(* Logix 5000 project; controller cal1615 1756-L62 rev 20.19; software revision 20.05; part 61 of 82 *)
(* tags used below, declared in another part *)
   aaa_eb_temp2 : BOOL;
   FAULT : BOOL;   // Fault AFI
   p01_recipe_active : recipe;   // Active Recipe
   p01r02_plc_scan_time_in_sec : REAL;   // System PLC Scan Time in Seconds
   p01r09_pb_global_reset : BOOL;   // System Modes PB: Global Fault Reset
   p01r09_request_line_jog : BOOL;   // System Modes Request Line Jog Forward
   p01r09_stretch_mode : BOOL;
   p01r12_master_ramped_speed : REAL;   // System Line Accel Decel Control Master Ramped Speed
   p01r13_line_running : BOOL;   // System Line Start Sequence Line Running
   p01r13_line_slow_ramp : BOOL;   // System Line Start Sequence Start Line to Slow Speed
   p01r13_permissive_drives : BOOL;   // System Line Start Sequence Permissive Drives
   p01r13_state : DINT;   // System Line Start Sequence Sequencer Step
   p02_real_from_hmi : hmi_real;   // MOP HMI Iface Real from HMI
   p20r15_loa_on : BOOL;   // Letoff Letoff A VFD On
   p20r16_lob_on : BOOL;   // Letoff Letoff B On
   p22r09_mode_thread : BOOL;   // Tension Stand 1 Modes Thread Mode
   p22r10_pid_psn : PID;   // Tension Stand 1 Speed Tension PID Dancer Position
   p25_ai_speed : REAL;   // Tension Stand 2 Inputs Sufrace Speed [fpm]
   p25_ai_torque : REAL;
   p25_ai_ts2_lc : REAL;   // System Metering Roll VFD Minimum Start Tension
   p25_ao_selected_speed : REAL;   // Tension Stand 2 VFD Selected Speed
   p25_ao_torque : REAL;
   p25_control_word : INT;
   p25_di_brake : BOOL;   // Tension Stand 2 Digital Input TS2 & Slitter Brake Temperature OK
   p25_di_therm : BOOL;   // Tension Stand 2 Digital Input Motor Temperature OK
   p25_param_ts2_jog_speed : REAL;   // System Parameter Tension Stand 2 Jog Speed
   p25_status_word : INT;
   p25_ts2_acc_rate : REAL;
   p25_ts2_decel_rate : REAL;
   p25_ts2_vfd : ABB_PROTOCOL_VFD;
   p25r01 : routine;
   p25r02_tension_dev_max : REAL;
   p25r02_tension_dev_min : REAL;
   p25r09_mode_jog : BOOL;   // Tension Stand 2 Modes Jog Mode
   p25r09_mode_thread : BOOL;   // Tension Stand 2 Modes Thread Mode
   p25r09_pb_jog_fwd : BOOL;   // Tension Stand 2 Modes PB: Jog Forward
   p25r09_pb_jog_rev : BOOL;   // Tension Stand 2 Modes PB: Jog Reverse
   p25r10 : routine;
   p25r10_calc_speed_offset : REAL;
   p25r10_param_psn_gain : REAL;   // Tension Stand 2 Parameter Position Gain
   p25r10_pid_manual_request : BOOL;
   p25r10_pid_out : REAL;
   p25r10_pid_psn : PID;   // Tension Stand 2 Speed Tension PID Dancer Position Process Variable
   p25r10_pid_psn_cv : REAL;
   p25r10_pid_psn_pv : REAL;   // Tension Stand 2 Speed Tension PID Dancer Position Process Variable
   p25r10_speed_offset : REAL;   // Tension Stand 2 Speed tension Speed Offset from Base
   p25r10_tension_request : BOOL;
   p25r10_timer_fault : TIMER[4];   // Tension Stand 2 Speed Tension Fault Dwell Timer
   p25r10_timer_warning : TIMER[4];   // Tension Stand 2 Speed Tension Warning Dwell Timer
   p25r11 : routine;   // Tension Stand 2 VFD
   p25r11_acc_decel_ramp : SYS_ACC_DEC_RAMP;   // Tension Stand 2 VFD Accel /Decel Ramp
   p25r11_at_zero : BOOL;   // Tension Stand 2 VFD At Zero Speed
   p25r11_permissive_jog_thread : BOOL;   // Tension Stand 2 VFD Permissive Jog/Thread
   p25r11_request_jog_fwd : BOOL;   // Tension Stand 2 VFD Request Jog FWD
   p25r11_request_jog_rev : BOOL;   // Tension Stand 2 VFD Request Jog REV
   p25r11_request_line_jog : BOOL;   // Tension Stand 2 VFD Request Line Jog
   p25r11_request_line_run : BOOL;   // Tension Stant 2 VFD Request Line Run
   p25r11_request_thread_fwd : BOOL;   // Tension Stand 2 VFD Request Thread FWD
   p25r11_request_thread_rev : BOOL;   // Tension Stand 2 VFD Request Thread REV
   p25r11_selected_speed : REAL;   // Tension Stand 2 VFD Selected Speed
   p25r11_timer_fault : TIMER[10];   // Tension Stand 2 VFD Fault Dwell Timer
   p25r11_timer_warning : TIMER[4];   // Tension Stand VFD Warning Dwell Timer
   p25r11_vfd_start_request : BOOL;
   p29r15 : routine;   // Winder Winder A VFD
(* P25_Tension_Stand_2, continued *)

ROUTINE R10_Speed_Control   (* ladder *)
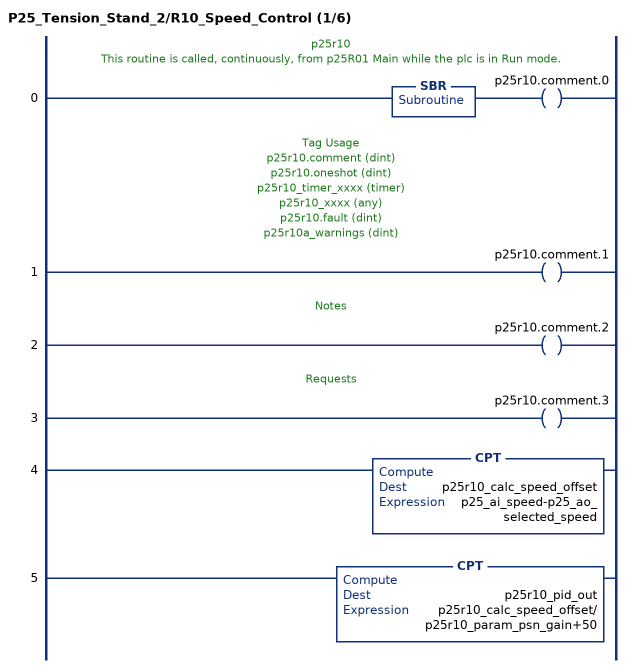
   // p25r10
   // This routine is called, continuously, from p25R01 Main while the plc is in Run mode.
   0: SBR()OTE(p25r10.comment.0);
   // Tag Usage
   // p25r10.comment (dint)
   // p25r10.oneshot (dint)
   // p25r10_timer_xxxx (timer)
   // p25r10_xxxx (any)
   // p25r10.fault (dint)
   // p25r10a_warnings (dint)
   1: OTE(p25r10.comment.1);
   // Notes
   2: OTE(p25r10.comment.2);
   // Requests
   3: OTE(p25r10.comment.3);
   4: CPT(p25r10_calc_speed_offset,p25_ai_speed-p25_ao_selected_speed);
   5: CPT(p25r10_pid_out,p25r10_calc_speed_offset/p25r10_param_psn_gain+50);
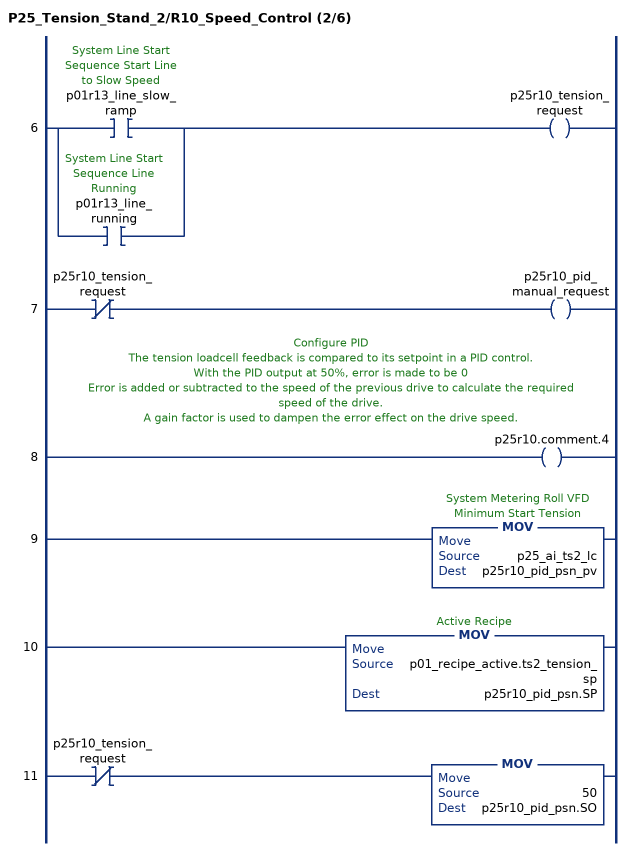
   6: [XIC(p01r13_line_slow_ramp) ,XIC(p01r13_line_running) ]OTE(p25r10_tension_request);
   7: XIO(p25r10_tension_request)OTE(p25r10_pid_manual_request);
   // Configure PID
   // The tension loadcell feedback is compared to its setpoint in a PID control.
   // With the PID output at 50%, error is made to be 0
   // Error is added or subtracted to the speed of the previous drive to calculate the required speed of the drive.
   // A gain factor is used to dampen the error effect on the drive speed.
   8: OTE(p25r10.comment.4);
   9: MOV(p25_ai_ts2_lc,p25r10_pid_psn_pv);
   10: MOV(p01_recipe_active.ts2_tension_sp,p25r10_pid_psn.SP);
   11: XIO(p25r10_tension_request)MOV(50,p25r10_pid_psn.SO);
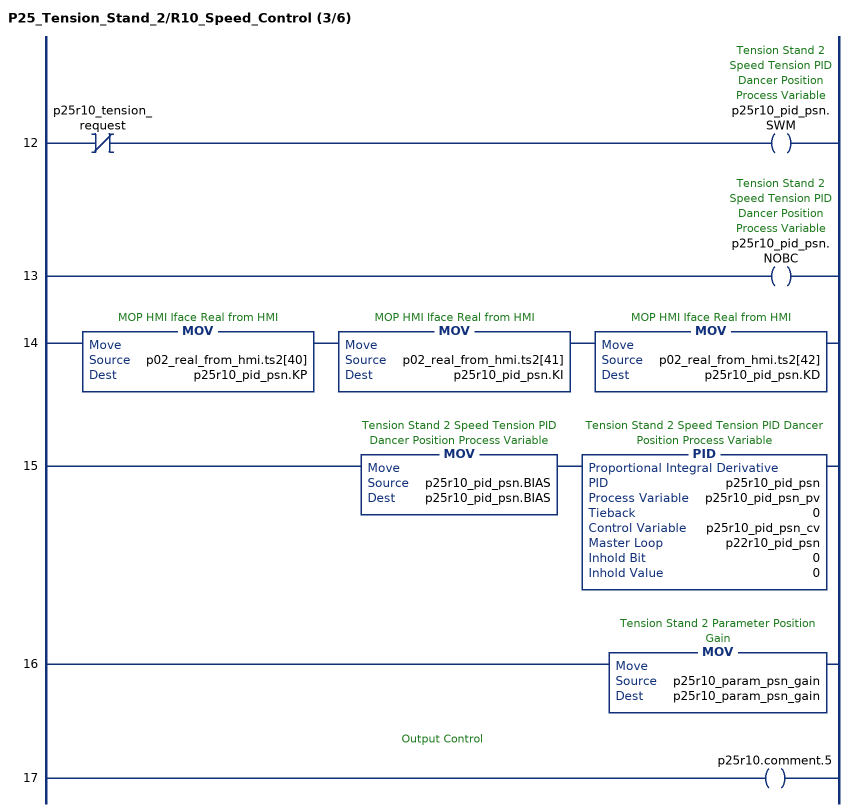
   12: XIO(p25r10_tension_request)OTE(p25r10_pid_psn.SWM);
   13: OTE(p25r10_pid_psn.NOBC);
   14: MOV(p02_real_from_hmi.ts2[40],p25r10_pid_psn.KP)MOV(p02_real_from_hmi.ts2[41],p25r10_pid_psn.KI)MOV(p02_real_from_hmi.ts2[42],p25r10_pid_psn.KD);
   15: MOV(p25r10_pid_psn.BIAS,p25r10_pid_psn.BIAS)PID(p25r10_pid_psn,p25r10_pid_psn_pv,0,p25r10_pid_psn_cv,p22r10_pid_psn,0,0);
   16: MOV(p25r10_param_psn_gain,p25r10_param_psn_gain);
   // Output Control
   17: OTE(p25r10.comment.5);
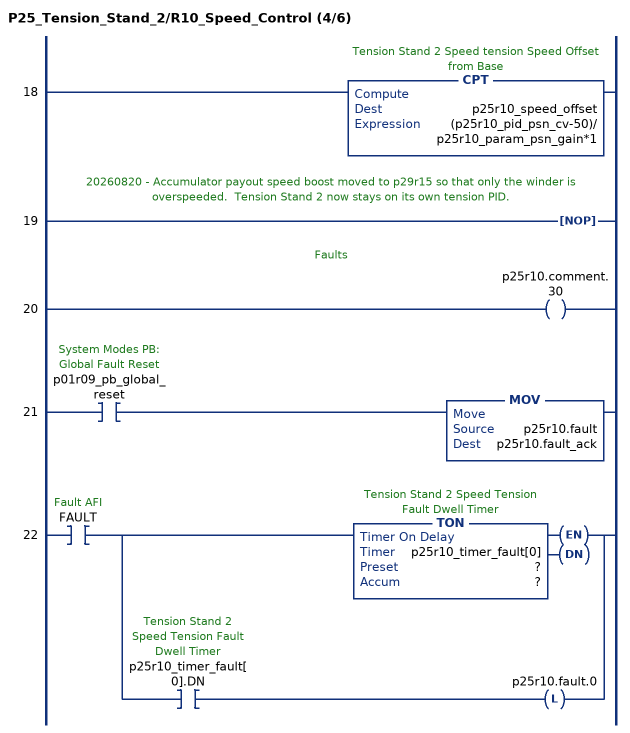
   18: CPT(p25r10_speed_offset,(p25r10_pid_psn_cv-50)/p25r10_param_psn_gain*1);
   // 20260820 - Accumulator payout speed boost moved to p29r15 so that only the winder is overspeeded.  Tension Stand 2 now stays on its own tension PID.
   19: NOP();
   // Faults
   20: OTE(p25r10.comment.30);
   21: XIC(p01r09_pb_global_reset)MOV(p25r10.fault,p25r10.fault_ack);
   22: XIC(FAULT)[TON(p25r10_timer_fault[0],?,?) ,XIC(p25r10_timer_fault[0].DN) OTL(p25r10.fault.0) ];
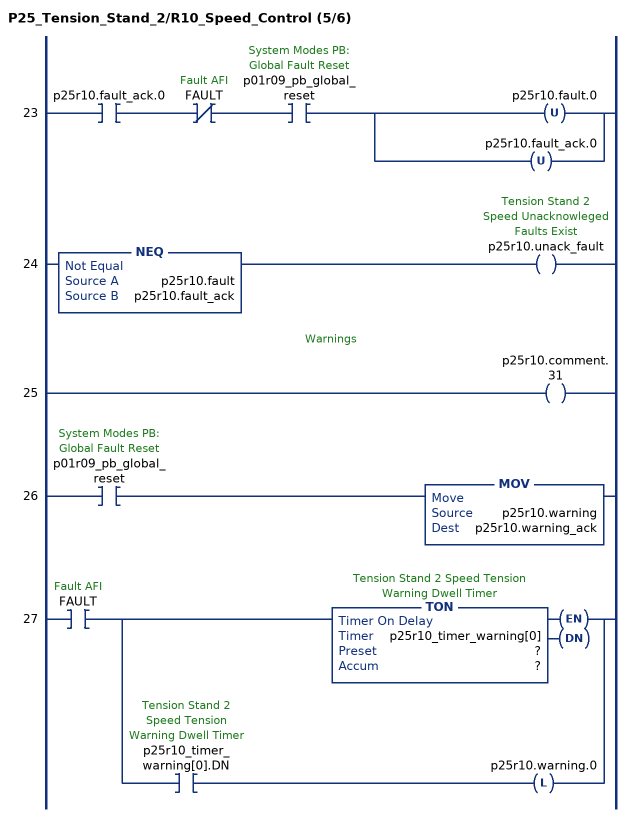
   23: XIC(p25r10.fault_ack.0)XIO(FAULT)XIC(p01r09_pb_global_reset)[OTU(p25r10.fault.0) ,OTU(p25r10.fault_ack.0) ];
   24: NEQ(p25r10.fault,p25r10.fault_ack)OTE(p25r10.unack_fault);
   // Warnings
   25: OTE(p25r10.comment.31);
   26: XIC(p01r09_pb_global_reset)MOV(p25r10.warning,p25r10.warning_ack);
   27: XIC(FAULT)[TON(p25r10_timer_warning[0],?,?) ,XIC(p25r10_timer_warning[0].DN) OTL(p25r10.warning.0) ];
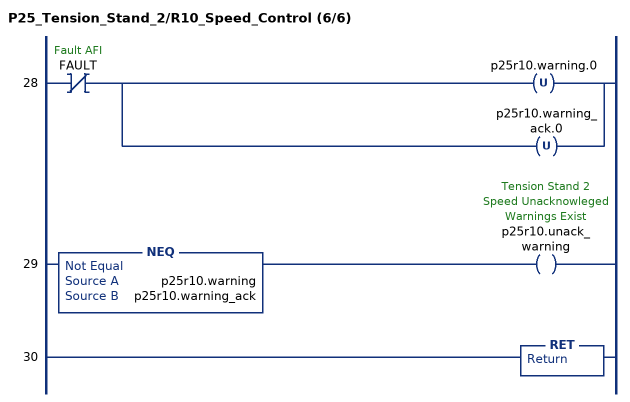
   28: XIO(FAULT)[OTU(p25r10.warning.0) ,OTU(p25r10.warning_ack.0) ];
   29: NEQ(p25r10.warning,p25r10.warning_ack)OTE(p25r10.unack_warning);
   30: RET();
END_ROUTINE

ROUTINE R11_VFD   (* ladder *)
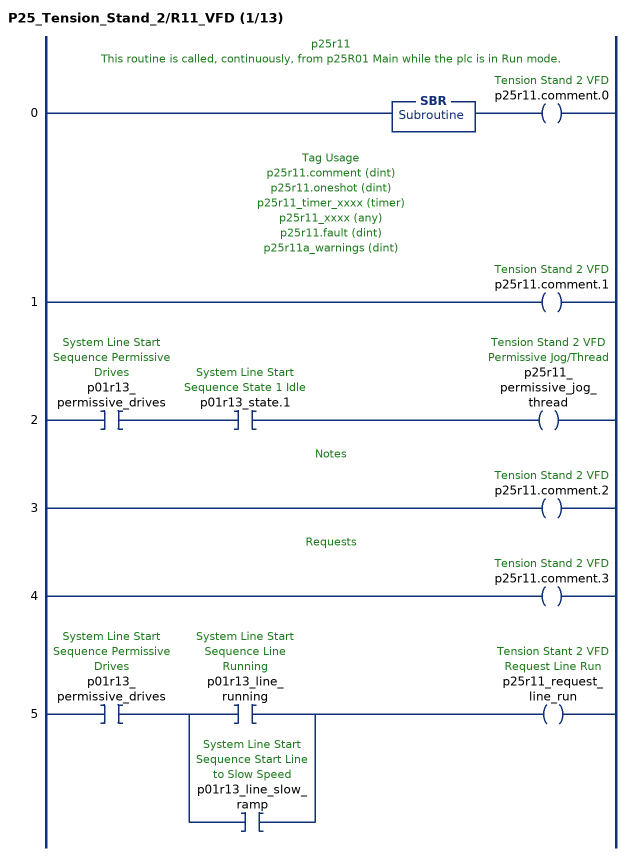
   // p25r11
   // This routine is called, continuously, from p25R01 Main while the plc is in Run mode.
   0: SBR()OTE(p25r11.comment.0);
   // Tag Usage
   // p25r11.comment (dint)
   // p25r11.oneshot (dint)
   // p25r11_timer_xxxx (timer)
   // p25r11_xxxx (any)
   // p25r11.fault (dint)
   // p25r11a_warnings (dint)
   1: OTE(p25r11.comment.1);
   2: XIC(p01r13_permissive_drives)XIC(p01r13_state.1)OTE(p25r11_permissive_jog_thread);
   // Notes
   3: OTE(p25r11.comment.2);
   // Requests
   4: OTE(p25r11.comment.3);
   5: XIC(p01r13_permissive_drives)[XIC(p01r13_line_running) ,XIC(p01r13_line_slow_ramp) ]OTE(p25r11_request_line_run);
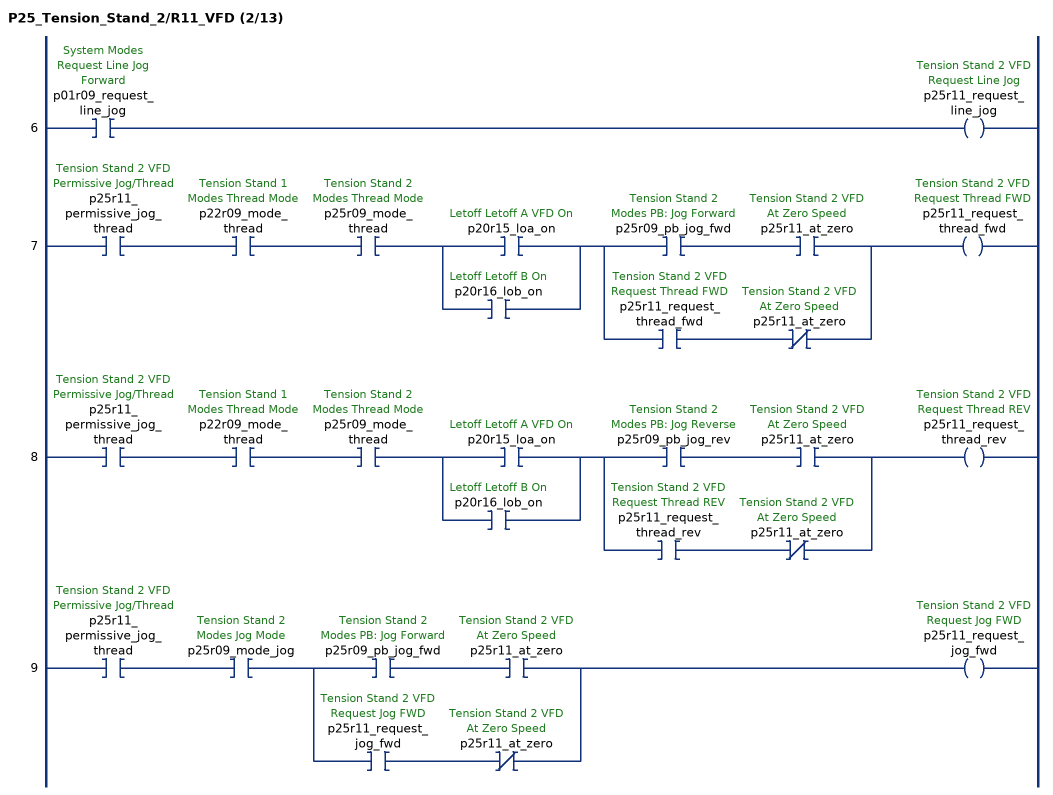
   6: XIC(p01r09_request_line_jog)OTE(p25r11_request_line_jog);
   7: XIC(p25r11_permissive_jog_thread)XIC(p22r09_mode_thread)XIC(p25r09_mode_thread)[XIC(p20r15_loa_on) ,XIC(p20r16_lob_on) ][XIC(p25r09_pb_jog_fwd) XIC(p25r11_at_zero) ,XIC(p25r11_request_thread_fwd) XIO(p25r11_at_zero) ]OTE(p25r11_request_thread_fwd);
   8: XIC(p25r11_permissive_jog_thread)XIC(p22r09_mode_thread)XIC(p25r09_mode_thread)[XIC(p20r15_loa_on) ,XIC(p20r16_lob_on) ][XIC(p25r09_pb_jog_rev) XIC(p25r11_at_zero) ,XIC(p25r11_request_thread_rev) XIO(p25r11_at_zero) ]OTE(p25r11_request_thread_rev);
   9: XIC(p25r11_permissive_jog_thread)XIC(p25r09_mode_jog)[XIC(p25r09_pb_jog_fwd) XIC(p25r11_at_zero) ,XIC(p25r11_request_jog_fwd) XIO(p25r11_at_zero) ]OTE(p25r11_request_jog_fwd);
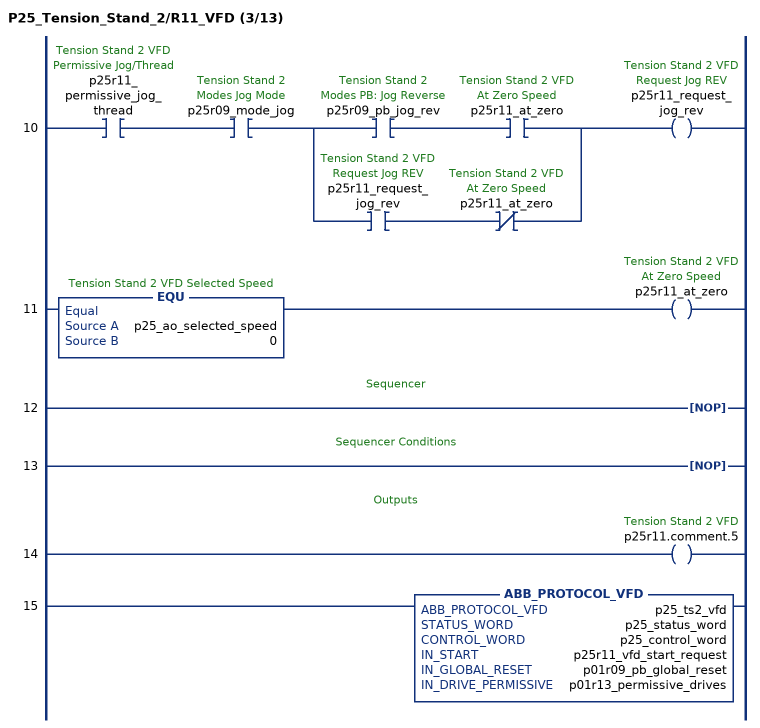
   10: XIC(p25r11_permissive_jog_thread)XIC(p25r09_mode_jog)[XIC(p25r09_pb_jog_rev) XIC(p25r11_at_zero) ,XIC(p25r11_request_jog_rev) XIO(p25r11_at_zero) ]OTE(p25r11_request_jog_rev);
   11: EQU(p25_ao_selected_speed,0)OTE(p25r11_at_zero);
   // Sequencer
   12: NOP();
   // Sequencer Conditions
   13: NOP();
   // Outputs
   14: OTE(p25r11.comment.5);
   15: ABB_PROTOCOL_VFD(p25_ts2_vfd,p25_status_word,p25_control_word,p25r11_vfd_start_request,p01r09_pb_global_reset,p01r13_permissive_drives);
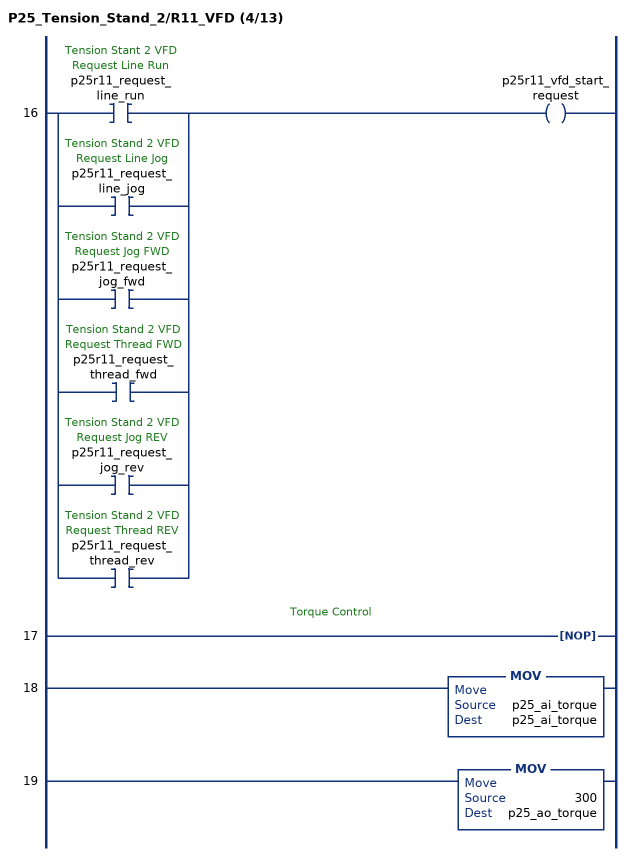
   16: [XIC(p25r11_request_line_run) ,XIC(p25r11_request_line_jog) ,XIC(p25r11_request_jog_fwd) ,XIC(p25r11_request_thread_fwd) ,XIC(p25r11_request_jog_rev) ,XIC(p25r11_request_thread_rev) ]OTE(p25r11_vfd_start_request);
   // Torque Control
   17: NOP();
   18: MOV(p25_ai_torque,p25_ai_torque);
   19: MOV(300,p25_ao_torque);
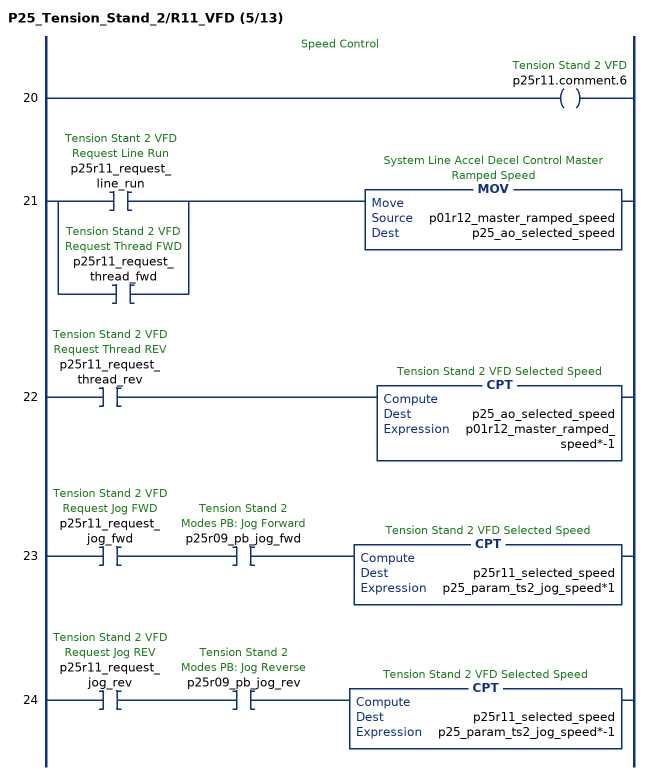
   // Speed Control
   20: OTE(p25r11.comment.6);
   21: [XIC(p25r11_request_line_run) ,XIC(p25r11_request_thread_fwd) ]MOV(p01r12_master_ramped_speed,p25_ao_selected_speed);
   22: XIC(p25r11_request_thread_rev)CPT(p25_ao_selected_speed,p01r12_master_ramped_speed*-1);
   23: XIC(p25r11_request_jog_fwd)XIC(p25r09_pb_jog_fwd)CPT(p25r11_selected_speed,p25_param_ts2_jog_speed*1);
   24: XIC(p25r11_request_jog_rev)XIC(p25r09_pb_jog_rev)CPT(p25r11_selected_speed,p25_param_ts2_jog_speed*-1);
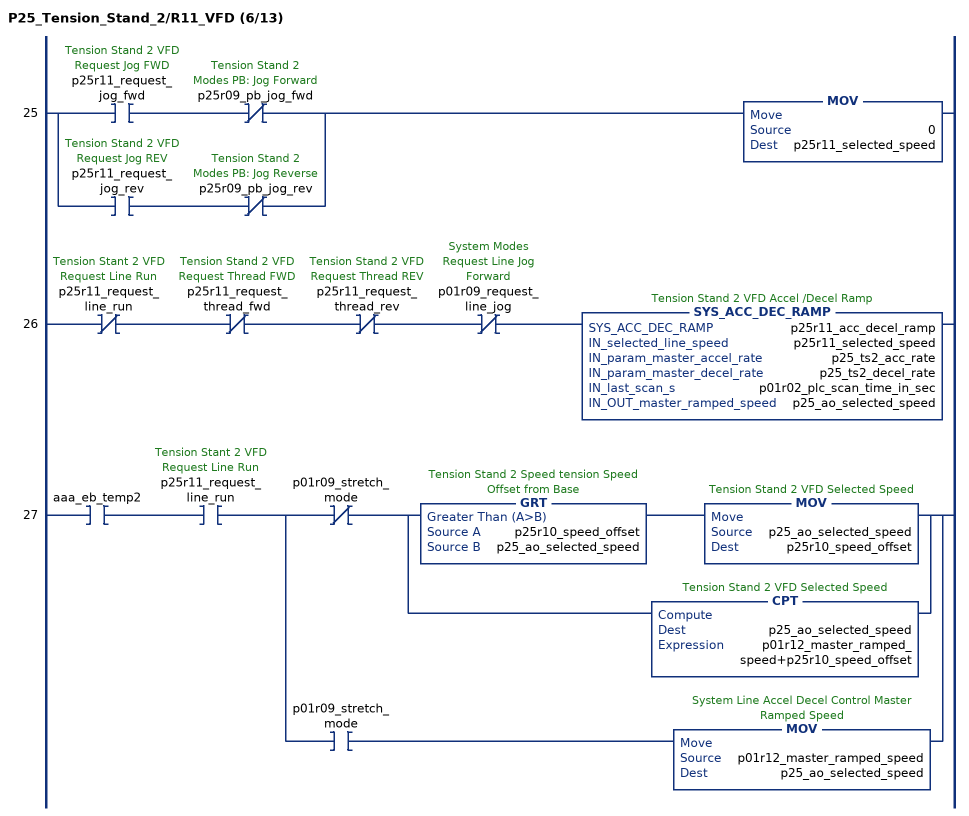
   25: [XIC(p25r11_request_jog_fwd) XIO(p25r09_pb_jog_fwd) ,XIC(p25r11_request_jog_rev) XIO(p25r09_pb_jog_rev) ]MOV(0,p25r11_selected_speed);
   26: XIO(p25r11_request_line_run)XIO(p25r11_request_thread_fwd)XIO(p25r11_request_thread_rev)XIO(p01r09_request_line_jog)SYS_ACC_DEC_RAMP(p25r11_acc_decel_ramp,p25r11_selected_speed,p25_ts2_acc_rate,p25_ts2_decel_rate,p01r02_plc_scan_time_in_sec,p25_ao_selected_speed);
   27: XIC(aaa_eb_temp2)XIC(p25r11_request_line_run)[XIO(p01r09_stretch_mode) [GRT(p25r10_speed_offset,p25_ao_selected_speed) MOV(p25_ao_selected_speed,p25r10_speed_offset) ,CPT(p25_ao_selected_speed,p01r12_master_ramped_speed+p25r10_speed_offset) ] ,XIC(p01r09_stretch_mode) MOV(p01r12_master_ramped_speed,p25_ao_selected_speed) ];
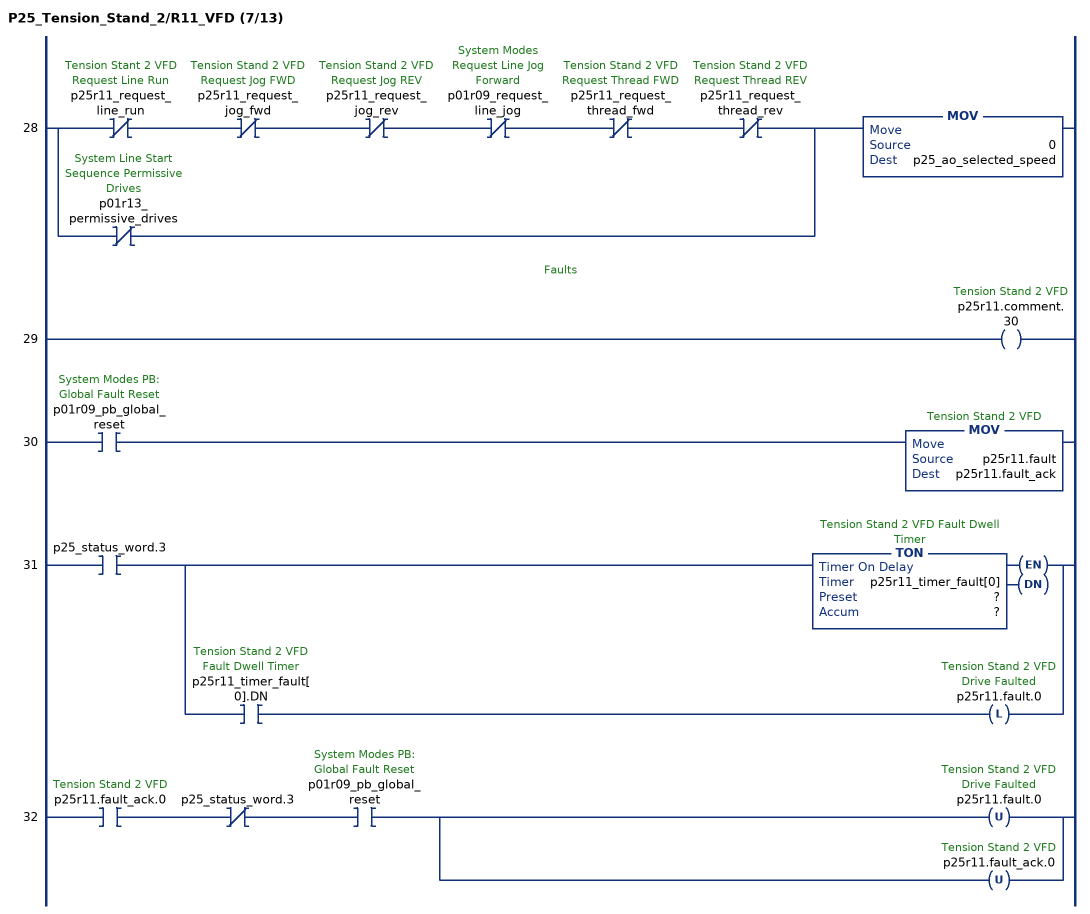
   28: [XIO(p25r11_request_line_run) XIO(p25r11_request_jog_fwd) XIO(p25r11_request_jog_rev) XIO(p01r09_request_line_jog) XIO(p25r11_request_thread_fwd) XIO(p25r11_request_thread_rev) ,XIO(p01r13_permissive_drives) ]MOV(0,p25_ao_selected_speed);
   // Faults
   29: OTE(p25r11.comment.30);
   30: XIC(p01r09_pb_global_reset)MOV(p25r11.fault,p25r11.fault_ack);
   31: XIC(p25_status_word.3)[TON(p25r11_timer_fault[0],?,?) ,XIC(p25r11_timer_fault[0].DN) OTL(p25r11.fault.0) ];
   32: XIC(p25r11.fault_ack.0)XIO(p25_status_word.3)XIC(p01r09_pb_global_reset)[OTU(p25r11.fault.0) ,OTU(p25r11.fault_ack.0) ];
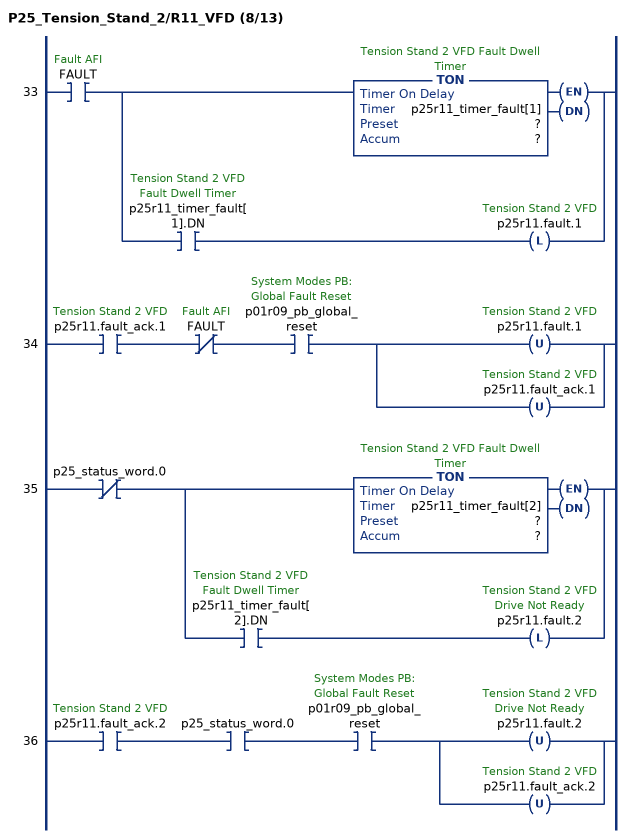
   33: XIC(FAULT)[TON(p25r11_timer_fault[1],?,?) ,XIC(p25r11_timer_fault[1].DN) OTL(p25r11.fault.1) ];
   34: XIC(p25r11.fault_ack.1)XIO(FAULT)XIC(p01r09_pb_global_reset)[OTU(p25r11.fault.1) ,OTU(p25r11.fault_ack.1) ];
   35: XIO(p25_status_word.0)[TON(p25r11_timer_fault[2],?,?) ,XIC(p25r11_timer_fault[2].DN) OTL(p25r11.fault.2) ];
   36: XIC(p25r11.fault_ack.2)XIC(p25_status_word.0)XIC(p01r09_pb_global_reset)[OTU(p25r11.fault.2) ,OTU(p25r11.fault_ack.2) ];
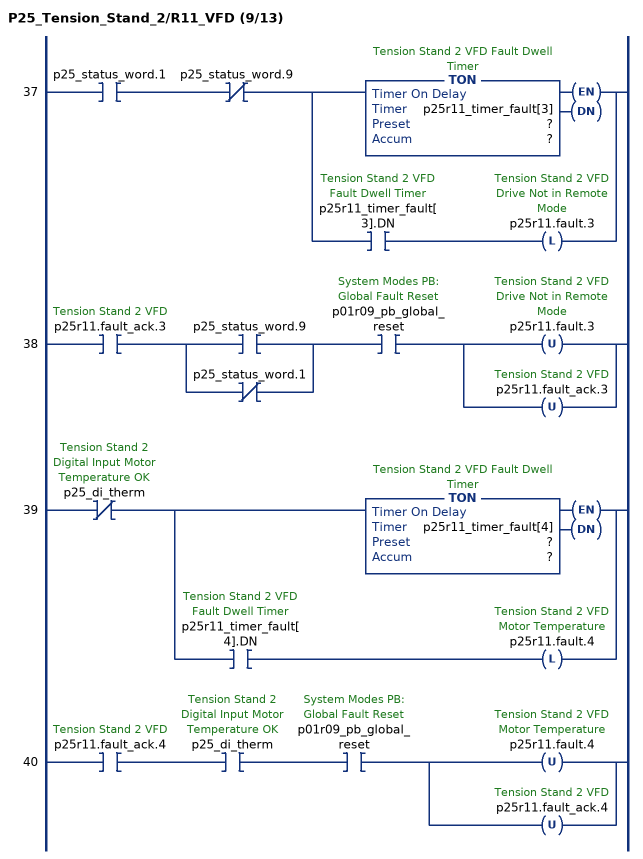
   37: XIC(p25_status_word.1)XIO(p25_status_word.9)[TON(p25r11_timer_fault[3],?,?) ,XIC(p25r11_timer_fault[3].DN) OTL(p25r11.fault.3) ];
   38: XIC(p25r11.fault_ack.3)[XIC(p25_status_word.9) ,XIO(p25_status_word.1) ]XIC(p01r09_pb_global_reset)[OTU(p25r11.fault.3) ,OTU(p25r11.fault_ack.3) ];
   39: XIO(p25_di_therm)[TON(p25r11_timer_fault[4],?,?) ,XIC(p25r11_timer_fault[4].DN) OTL(p25r11.fault.4) ];
   40: XIC(p25r11.fault_ack.4)XIC(p25_di_therm)XIC(p01r09_pb_global_reset)[OTU(p25r11.fault.4) ,OTU(p25r11.fault_ack.4) ];
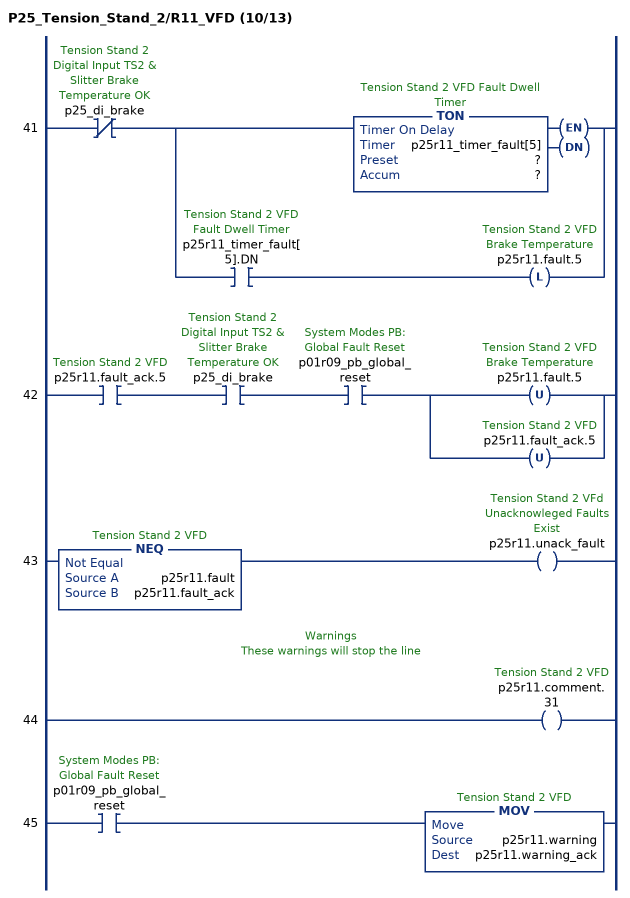
   41: XIO(p25_di_brake)[TON(p25r11_timer_fault[5],?,?) ,XIC(p25r11_timer_fault[5].DN) OTL(p25r11.fault.5) ];
   42: XIC(p25r11.fault_ack.5)XIC(p25_di_brake)XIC(p01r09_pb_global_reset)[OTU(p25r11.fault.5) ,OTU(p25r11.fault_ack.5) ];
   43: NEQ(p25r11.fault,p25r11.fault_ack)OTE(p25r11.unack_fault);
   // Warnings
   // These warnings will stop the line
   44: OTE(p25r11.comment.31);
   45: XIC(p01r09_pb_global_reset)MOV(p25r11.warning,p25r11.warning_ack);
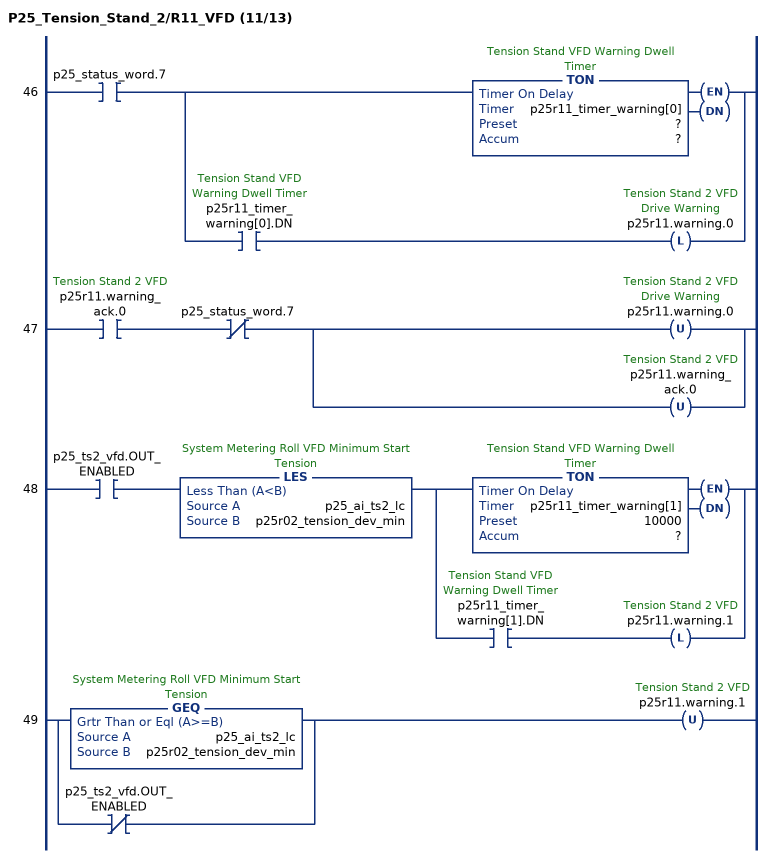
   46: XIC(p25_status_word.7)[TON(p25r11_timer_warning[0],?,?) ,XIC(p25r11_timer_warning[0].DN) OTL(p25r11.warning.0) ];
   47: XIC(p25r11.warning_ack.0)XIO(p25_status_word.7)[OTU(p25r11.warning.0) ,OTU(p25r11.warning_ack.0) ];
   48: XIC(p25_ts2_vfd.OUT_ENABLED)LES(p25_ai_ts2_lc,p25r02_tension_dev_min)[TON(p25r11_timer_warning[1],?,?) ,XIC(p25r11_timer_warning[1].DN) OTL(p25r11.warning.1) ];
   49: [GEQ(p25_ai_ts2_lc,p25r02_tension_dev_min) ,XIO(p25_ts2_vfd.OUT_ENABLED) ]OTU(p25r11.warning.1);
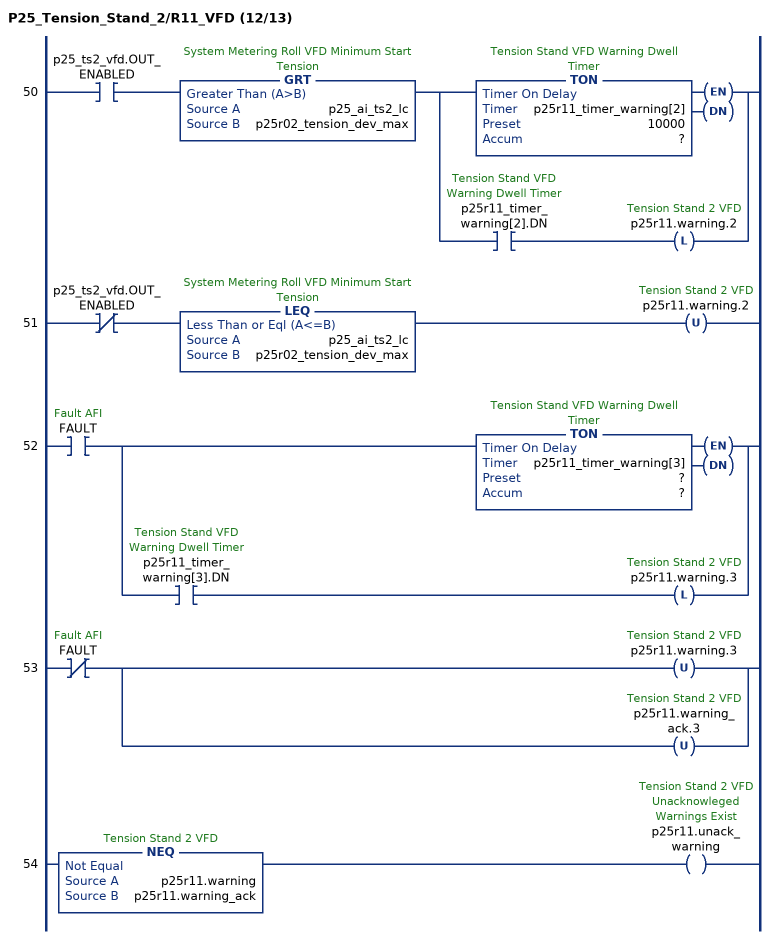
   50: XIC(p25_ts2_vfd.OUT_ENABLED)GRT(p25_ai_ts2_lc,p25r02_tension_dev_max)[TON(p25r11_timer_warning[2],?,?) ,XIC(p25r11_timer_warning[2].DN) OTL(p25r11.warning.2) ];
   51: XIO(p25_ts2_vfd.OUT_ENABLED)LEQ(p25_ai_ts2_lc,p25r02_tension_dev_max)OTU(p25r11.warning.2);
   52: XIC(FAULT)[TON(p25r11_timer_warning[3],?,?) ,XIC(p25r11_timer_warning[3].DN) OTL(p25r11.warning.3) ];
   53: XIO(FAULT)[OTU(p25r11.warning.3) ,OTU(p25r11.warning_ack.3) ];
   54: NEQ(p25r11.warning,p25r11.warning_ack)OTE(p25r11.unack_warning);
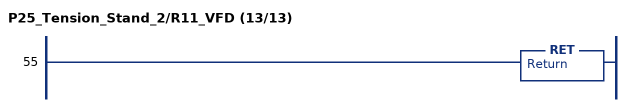
   55: RET();
END_ROUTINE
END_PROGRAM
